{attribute 'qualified_only'}
TYPE E_State :
(
	Init := 0,
	ReadOnce,
	Error,
	Idle,
	Wait

	
);
END_TYPE

(* stored: Version 1.1.0.1, ProductVersion 3.1.4024.12
   DUT E_State: Id {152610e0-cdbf-4e25-93df-dac94cd9b39b} *)
